Omron CX-Programmer project NewProject (CX-Programmer 9.03)

# PLC NewPLC1: CJ1M CPU11
; 
I/O table (CPU CJ1M-CPU11): rack 0 slot 0 CJ1W-ID211; rack 0 slot 1 CJ1W-OC211; rack 0 slot 2 CJ1W-ID211; rack 0 slot 3 CJ1W-ID211

## Global symbols (name address type ; comment)
C0001 BOOL  ; Za 30 stepeni
C0003 BOOL  ; Za 60 stepeni
C0004 BOOL  ; Za 90 stepeni
T0001 BOOL  ; Vreme punjenja masine vodom
T0004 BOOL  ; Bubanj se okrece levo
T0005 BOOL  ; Pauza
T0006 BOOL  ; Motor se okrece desno

## Program NewProgram1 (cyclic task 0)
Local symbols
Centrifuga 2960.11 BOOL  ; Paljenje motora za centrifugu
Flag1 200.01 BOOL
Flag10 200.10 BOOL
Flag11 200.11 BOOL
Flag12 200.12 BOOL
Flag13 200.13 BOOL
Flag14 200.14 BOOL
Flag15 200.15 BOOL
Flag16 200.00 BOOL
Flag17 201.00 BOOL
Flag18 201.01 BOOL
Flag2 200.02 BOOL
Flag3 200.03 BOOL
Flag4 200.04 BOOL
Flag5 200.05 BOOL
Flag6 200.06 BOOL
Flag7 200.07 BOOL
Flag8 200.08 BOOL
Flag9 200.09 BOOL
Grejac 2961.04 BOOL
Lampica_kraj 2961.00 BOOL
Lampica_omeksivac 2961.09 BOOL  ; U toku je uzimanje omeksivaca
Lampica_prasak 2961.08 BOOL  ; U toku je uzimanje praska
Lampica_start 2961.03 BOOL
MotorDesno 2961.02 BOOL  ; Bubanj se okrece na desno
MotorLevo 2961.01 BOOL  ; Bubanj se okrece na levo
Pauza 2960.14 BOOL  ; Pauza izmedju levo i desno
Pranje_desno 2960.13 BOOL  ; Bubanj se vrti u  desno
Pranje_levo 2960.12 BOOL  ; Bubanj se vrti u levo
PrekidacPamuk 2960.07 BOOL
PrekidacSintetika 2960.08 BOOL
PrekidacVuna 2960.09 BOOL
Prekidac_30s 2960.04 BOOL
Prekidac_60s 2960.05 BOOL
Prekidac_90s 2960.06 BOOL
Pumpa1 2961.10 BOOL  ; Ubacuje se voda u bubanj
Pumpa2 2960.15 BOOL  ; Pumpa za izbacivanje vode iz masine
Senzor30 3960.02 BOOL  ; Temperaturni senzor do 30 stepeni
Senzor60 2961.11 BOOL  ; Temperaturni senzor do 60 stepeni
Senzor90 3960.01 BOOL  ; Temperaturni senzor do 90 stepeni
SenzorMotorDesno 2960.03 BOOL
SenzorMotorLevo 2960.01 BOOL
SenzorResetMotor 2960.00 BOOL
Senzor_vrata 3960.00 BOOL
Start 2960.02 BOOL
StopSenzorMotor 2960.10 BOOL
Ventil1 2961.06 BOOL  ; Ventil za uzimanje praska
Ventil2 2961.07 BOOL  ; Ventil za uzimanje omeksivaca
Vrata_zakljucavanje 2961.05 BOOL

### Section Section1

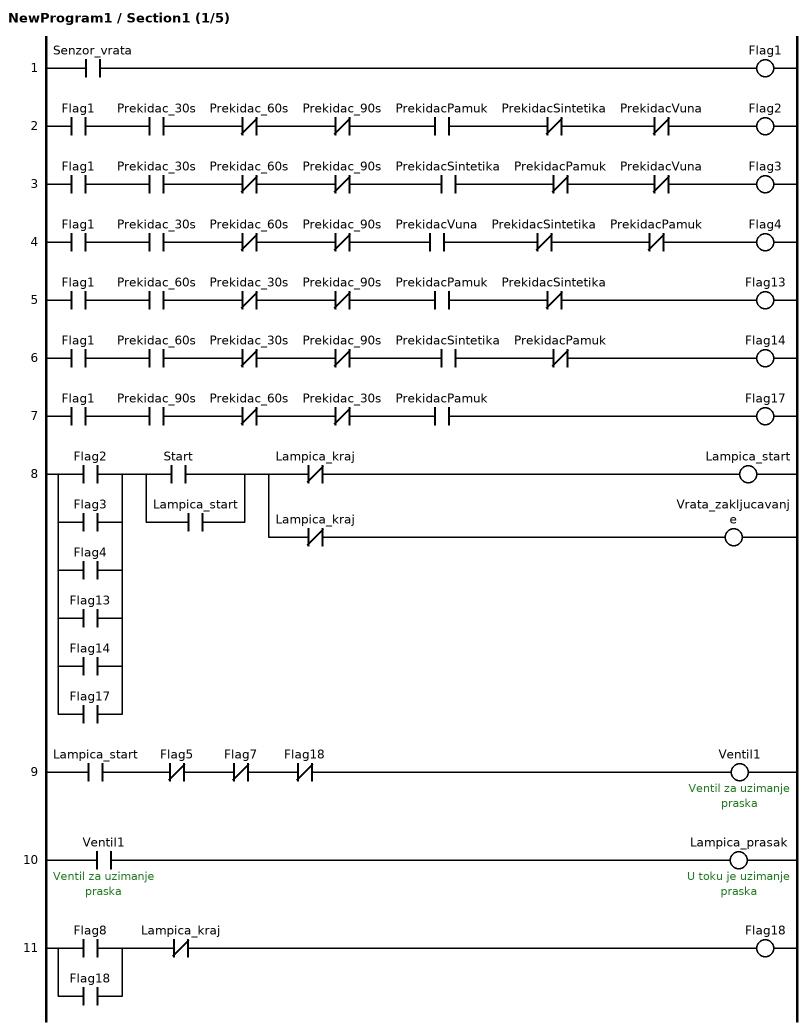
; rung 1
LD Senzor_vrata
OUT Flag1
; rung 2
LD Flag1
AND Prekidac_30s
ANDNOT Prekidac_60s
ANDNOT Prekidac_90s
AND PrekidacPamuk
ANDNOT PrekidacSintetika
ANDNOT PrekidacVuna
OUT Flag2
; rung 3
LD Flag1
AND Prekidac_30s
ANDNOT Prekidac_60s
ANDNOT Prekidac_90s
AND PrekidacSintetika
ANDNOT PrekidacPamuk
ANDNOT PrekidacVuna
OUT Flag3
; rung 4
LD Flag1
AND Prekidac_30s
ANDNOT Prekidac_60s
ANDNOT Prekidac_90s
AND PrekidacVuna
ANDNOT PrekidacSintetika
ANDNOT PrekidacPamuk
OUT Flag4
; rung 5
LD Flag1
AND Prekidac_60s
ANDNOT Prekidac_30s
ANDNOT Prekidac_90s
AND PrekidacPamuk
ANDNOT PrekidacSintetika
OUT Flag13
; rung 6
LD Flag1
AND Prekidac_60s
ANDNOT Prekidac_30s
ANDNOT Prekidac_90s
AND PrekidacSintetika
ANDNOT PrekidacPamuk
OUT Flag14
; rung 7
LD Flag1
AND Prekidac_90s
ANDNOT Prekidac_60s
ANDNOT Prekidac_30s
AND PrekidacPamuk
OUT Flag17
; rung 8
LD Flag2
OR Flag3
OR Flag4
OR Flag13
OR Flag14
OR Flag17
LD Start
OR Lampica_start
ANDLD
OUT TR0
ANDNOT Lampica_kraj
OUT Lampica_start
LD TR0
ANDNOT Lampica_kraj
OUT Vrata_zakljucavanje
; rung 9
LD Lampica_start
ANDNOT Flag5
ANDNOT Flag7
ANDNOT Flag18
OUT Ventil1  ; Ventil za uzimanje praska
; rung 10
LD Ventil1  ; Ventil za uzimanje praska
OUT Lampica_prasak  ; U toku je uzimanje praska
; rung 11
LD Flag8
OR Flag18
ANDNOT Lampica_kraj
OUT Flag18

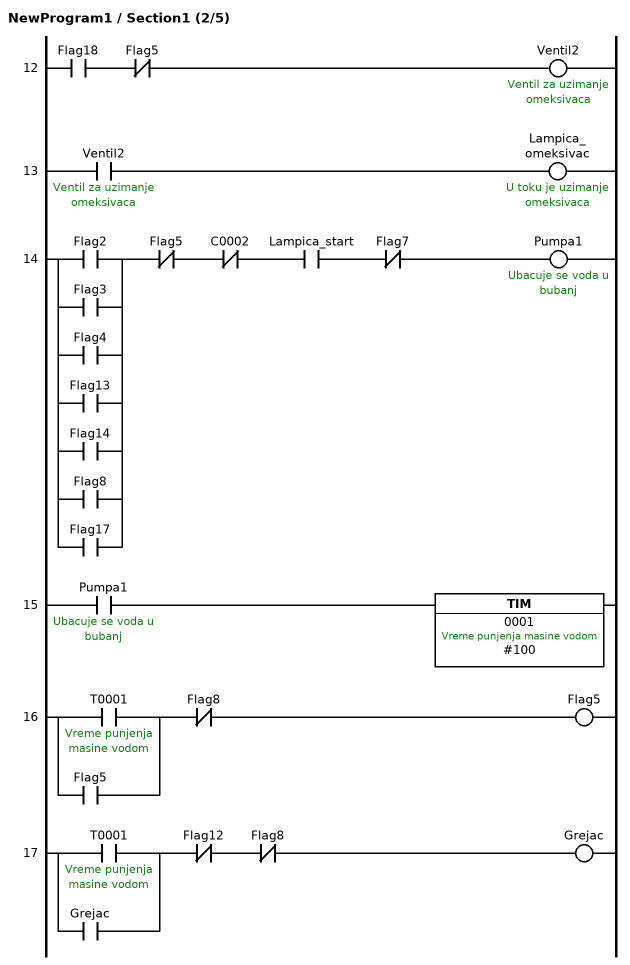
; rung 12
LD Flag18
ANDNOT Flag5
OUT Ventil2  ; Ventil za uzimanje omeksivaca
; rung 13
LD Ventil2  ; Ventil za uzimanje omeksivaca
OUT Lampica_omeksivac  ; U toku je uzimanje omeksivaca
; rung 14
LD Flag2
OR Flag3
OR Flag4
OR Flag13
OR Flag14
OR Flag8
OR Flag17
ANDNOT Flag5
ANDNOT C0002
AND Lampica_start
ANDNOT Flag7
OUT Pumpa1  ; Ubacuje se voda u bubanj
; rung 15
LD Pumpa1  ; Ubacuje se voda u bubanj
TIM 0001 #100  ; Vreme punjenja masine vodom
; rung 16
LD T0001  ; Vreme punjenja masine vodom
OR Flag5
ANDNOT Flag8
OUT Flag5
; rung 17
LD T0001  ; Vreme punjenja masine vodom
OR Grejac
ANDNOT Flag12
ANDNOT Flag8
OUT Grejac

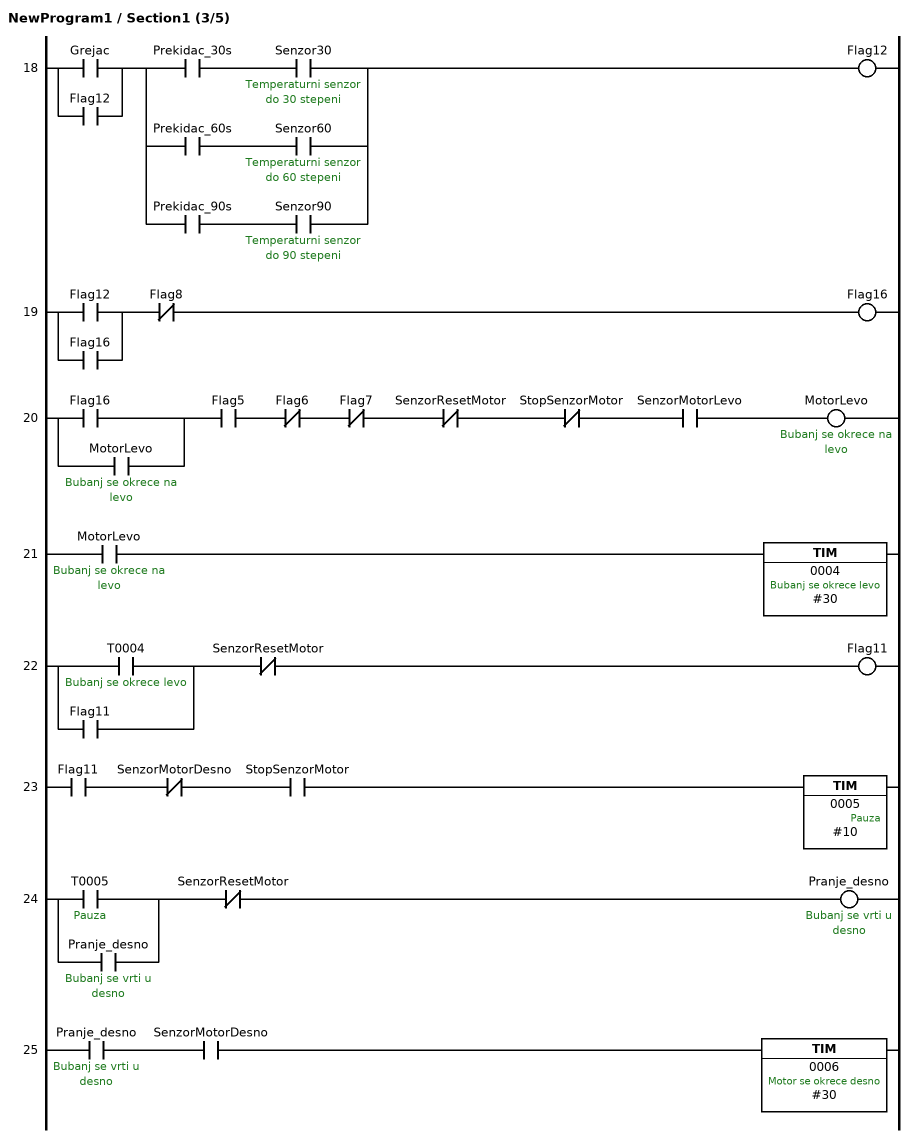
; rung 18
LD Grejac
OR Flag12
LD Prekidac_30s
AND Senzor30  ; Temperaturni senzor do 30 stepeni
LD Prekidac_60s
AND Senzor60  ; Temperaturni senzor do 60 stepeni
ORLD
LD Prekidac_90s
AND Senzor90  ; Temperaturni senzor do 90 stepeni
ORLD
ANDLD
OUT Flag12
; rung 19
LD Flag12
OR Flag16
ANDNOT Flag8
OUT Flag16
; rung 20
LD Flag16
OR MotorLevo  ; Bubanj se okrece na levo
AND Flag5
ANDNOT Flag6
ANDNOT Flag7
ANDNOT SenzorResetMotor
ANDNOT StopSenzorMotor
AND SenzorMotorLevo
OUT MotorLevo  ; Bubanj se okrece na levo
; rung 21
LD MotorLevo  ; Bubanj se okrece na levo
TIM 0004 #30  ; Bubanj se okrece levo
; rung 22
LD T0004  ; Bubanj se okrece levo
OR Flag11
ANDNOT SenzorResetMotor
OUT Flag11
; rung 23
LD Flag11
ANDNOT SenzorMotorDesno
AND StopSenzorMotor
TIM 0005 #10  ; Pauza
; rung 24
LD T0005  ; Pauza
OR Pranje_desno  ; Bubanj se vrti u  desno
ANDNOT SenzorResetMotor
OUT Pranje_desno  ; Bubanj se vrti u  desno
; rung 25
LD Pranje_desno  ; Bubanj se vrti u  desno
AND SenzorMotorDesno
TIM 0006 #30  ; Motor se okrece desno

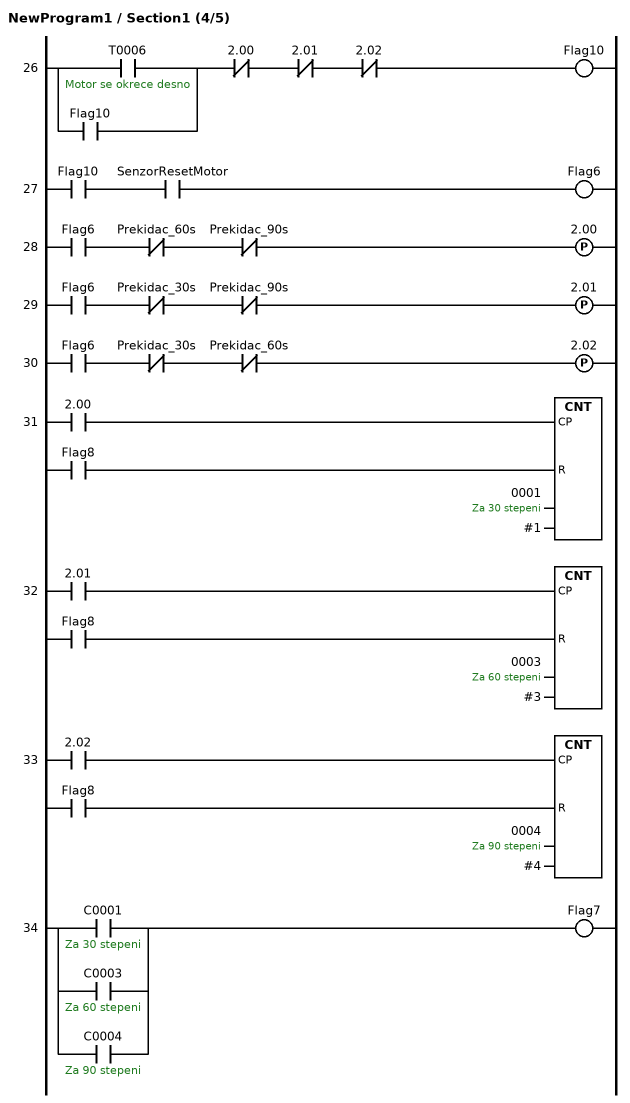
; rung 26
LD T0006  ; Motor se okrece desno
OR Flag10
ANDNOT 2.00
ANDNOT 2.01
ANDNOT 2.02
OUT Flag10
; rung 27
LD Flag10
AND SenzorResetMotor
OUT Flag6
; rung 28
LD Flag6
ANDNOT Prekidac_60s
ANDNOT Prekidac_90s
DIFU(013) 2.00
; rung 29
LD Flag6
ANDNOT Prekidac_30s
ANDNOT Prekidac_90s
DIFU(013) 2.01
; rung 30
LD Flag6
ANDNOT Prekidac_30s
ANDNOT Prekidac_60s
DIFU(013) 2.02
; rung 31
LD 2.00
LD Flag8
CNT 0001 #1  ; Za 30 stepeni
; rung 32
LD 2.01
LD Flag8
CNT 0003 #3  ; Za 60 stepeni
; rung 33
LD 2.02
LD Flag8
CNT 0004 #4  ; Za 90 stepeni
; rung 34
LD C0001  ; Za 30 stepeni
OR C0003  ; Za 60 stepeni
OR C0004  ; Za 90 stepeni
OUT Flag7

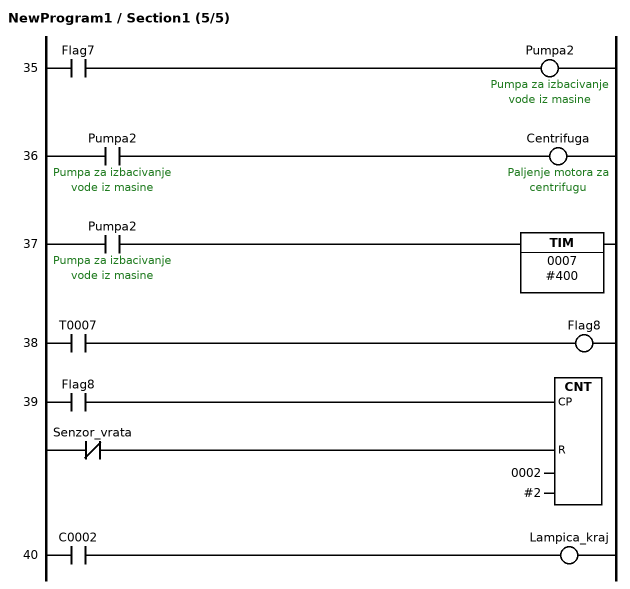
; rung 35
LD Flag7
OUT Pumpa2  ; Pumpa za izbacivanje vode iz masine
; rung 36
LD Pumpa2  ; Pumpa za izbacivanje vode iz masine
OUT Centrifuga  ; Paljenje motora za centrifugu
; rung 37
LD Pumpa2  ; Pumpa za izbacivanje vode iz masine
TIM 0007 #400
; rung 38
LD T0007
OUT Flag8
; rung 39
LD Flag8
LDNOT Senzor_vrata
CNT 0002 #2
; rung 40
LD C0002
OUT Lampica_kraj

### Section END
; rung 0
END(001)